INTERFACE SpindleController

// Return the current speed of the spindle in RPM
METHOD GetSpeed : UDINT
VAR_INPUT
END_VAR
END_METHOD

METHOD HasFault : BOOL
VAR_INPUT
END_VAR
END_METHOD

// Start the Spindle running
METHOD Run : BOOL
END_METHOD

// Set the direction the spindle rotates in.
METHOD SetDirection : BOOL
VAR_INPUT
	// Set the spindle rotation direction
	Reverse : BOOL;
END_VAR
END_METHOD

// Set the target speed for the spindle.
METHOD SetSpeed : BOOL
VAR_INPUT
	Speed : UINT;
END_VAR
END_METHOD

// Stop the running spindle
METHOD Stop : BOOL
END_METHOD

END_INTERFACE

(* stored: Version 1.1.0.1, ProductVersion 3.1.4022.17
   Itf SpindleController: Id {df9af8cd-f926-49bc-9ede-9a0faf189bc9}
   Method GetSpeed: Id {b7b1fee2-3c6f-4eca-abb5-cabb91af2c0d}
   Method HasFault: Id {3bd6f5ad-e08e-4f6f-8b38-2e578ebe5a92}
   Method Run: Id {bde1c9a9-ee7f-4e70-897d-f6e0e05beb6a}
   Method SetDirection: Id {34672ef6-92f0-4960-b735-ea7a89f86797}
   Method SetSpeed: Id {cb2af7f9-4e6c-4e88-9d58-7c04bcf58105}
   Method Stop: Id {775584b9-1b67-4b01-a066-f4712b5973a1} *)
